(* IEC 61131-3 sources: std_i2980_v2.06_cp053/Source/IMM/ieccontrol/Ejector1, 2 files *)

(* ---- ABMeasure.pu ---- *)
IMPORT_OVER_LISTFILE
 GET_MY_FU_NAME
, KSWO_AddVariable
, WRITE_SVREAL_DIRECT
, FAddToScopeGroup
, KAPPL_LintabData_2P
, KAPPL_MeasureMonitoring
, KSWO_Status
, ABMeasureAI

END_IMPORT

ALGORITHM_BLOCK ABMeasure #DUMMY_EDIT_BLOCK

SYSTEM_VAR
 sv_EjectorLintab : KAPPL_LintabData_2P;
 sv_rEjectorPosition : REAL;
 ai_Position : REAL;
 sv_bTransducerError : BOOL;
 sv_bDeviceReady : BOOL;
 sv_rEjectorVelocity : REAL;
 sv_EjectorMonitorMeas : KAPPL_MeasureMonitoring;
END_VAR

SYSTEM_OBJECT
 TaskAnalog : TASK;
 TaskSlow : TASK;
END_OBJECT

PROCESS_ALGORITHM paInitDebugMeasurement ON TaskSlow AUTOSTART

VAR
 variableName : STRING(255);
 swoState : KSWO_Status;
 b : BOOL;
END_VAR
#BEGIN_EDIT_BLOCK
(**************************************** WARNING ********************************************
 *** The KEBA Kemro K2 System including software is not intended for safety control tasks! ***
 ***                       For further information see Comment tab!                        ***
 *********************************************************************************************)

variableName := CONCAT(GET_MY_FU_NAME(),'.rPosition mm');
swoState := KSWO_AddVariable( Task := TaskAnalog,
                              Name := variableName,
                              Variable := sv_rEjectorPosition);
b := FAddToScopeGroup(Task := TaskAnalog,
                      Name := variableName,
                      GroupId := cScopeGroupEjector);
variableName := CONCAT(GET_MY_FU_NAME(),'.rVelocity mm/s');
swoState := KSWO_AddVariable( Task := TaskAnalog,
                              Name := variableName,
                              Variable := sv_rEjectorVelocity);
b := FAddToScopeGroup(Task := TaskAnalog,
                      Name := variableName,
                      GroupId := cScopeGroupEjector);

STOP_PROCESS_ALGORITHM();

;#END_EDIT_BLOCK END_ALGORITHM

PROCESS_ALGORITHM paMeasure ON TaskAnalog(1000) AUTOSTART

VAR_TEMP
 b : BOOL;
END_VAR

VAR
 abEjectorMeasure : ABMeasureAI;
END_VAR

(* IecGraph-Code *)

(* init step *)
INITIAL_STEP S_Start:
END_STEP

(* steps *)
STEP S_Stop:
AStop (P);
END_STEP

ACTION AStop: #BEGIN_EDIT_BLOCK
STOP_PROCESS_ALGORITHM();

;#END_EDIT_BLOCK END_ACTION (*AStop*)
STEP S_Init:
AInitMeasureBlock (P);
END_STEP

STEP S_Measure:
AMeasure (N);
END_STEP

(* transitions *)
TRANSITION TLinked (* TLinked *) FROM S_Start TO S_Init :=  #BEGIN_EDIT_BLOCK
IS_LINKED(ai_Position)
;#END_EDIT_BLOCK
END_TRANSITION

TRANSITION TNotLinked (* TNotLinked *) FROM S_Start TO S_Stop :=  #BEGIN_EDIT_BLOCK
NOT IS_LINKED(ai_Position)
;#END_EDIT_BLOCK
END_TRANSITION

TRANSITION TStop (* TStop *) FROM S_Stop TO S_Start :=  #BEGIN_EDIT_BLOCK
TRUE
;#END_EDIT_BLOCK
END_TRANSITION

TRANSITION TInitDone (* TInitDone *) FROM S_Init TO S_Measure :=  #BEGIN_EDIT_BLOCK
TRUE
;#END_EDIT_BLOCK
END_TRANSITION

(* end IecGraph-Code *)
(* sfc-code *)

(* stand alone actions *)
ACTION AMeasure: #BEGIN_EDIT_BLOCK
(**************************************** WARNING ********************************************
 *** The KEBA Kemro K2 System including software is not intended for safety control tasks! ***
 ***                       For further information see Comment tab!                        ***
 *********************************************************************************************)

abEjectorMeasure.aRun(bIdle := sv_bDeviceReady);
sv_bTransducerError := abEjectorMeasure.aRun.bSensorError;
b := WRITE_SVREAL_DIRECT(sv_rEjectorPosition, abEjectorMeasure.aRun.rValue);
b := WRITE_SVREAL_DIRECT(sv_rEjectorVelocity, abEjectorMeasure.aRun.rVelocity);

;#END_EDIT_BLOCK END_ACTION (*AMeasure*)
ACTION AInitMeasureBlock: #BEGIN_EDIT_BLOCK
(**************************************** WARNING ********************************************
 *** The KEBA Kemro K2 System including software is not intended for safety control tasks! ***
 ***                       For further information see Comment tab!                        ***
 *********************************************************************************************)

abEjectorMeasure.aInit(sRawValue := 'Ejector1.ai_Position',
                       pLintabPointArray :=  @sv_EjectorLintab.LintabPoints.Point,
                       piUsedLintabPoints := @sv_EjectorLintab.LintabPoints.uNoOfPoints);

abEjectorMeasure.aInitMonitoring(bEnable := sv_EjectorMonitorMeas.EnableMonitoring,
                                 rLowLimit := sv_EjectorMonitorMeas.LowerLimit,
                                 bLimitation := sv_EjectorMonitorMeas.Limitation,
                                 rFailureFactor := sv_EjectorMonitorMeas.FailureFactor);

;#END_EDIT_BLOCK END_ACTION (*AInitMeasureBlock*)
(* end sfc-code *)

END_ALGORITHM

END_ALGORITHM_BLOCK

#END_OF_IEC_PART

@Puma @IecEditor 6 103 @Pou 25
@@@BEG_Comment@@@

@@@END_Comment@@@

@BEG_Contents

@BEG_Func
@RT(17)FuncTreeContainer
4
@Var @RT(14)GET_MY_FU_NAME @RT(0) @T @T @DERIVED 0 @F @RT(22)KEBA_STANDARD_FUNCTION @F
@T
@BEG_Attrib
0 @RT(0) @RT(0)
@END_Attrib
1 1 @F @F @F @F

@Var @RT(16)KSWO_AddVariable @RT(0) @T @T @DERIVED 0 @F @RT(22)KEBA_STANDARD_FUNCTION @F
@T
@BEG_Attrib
0 @RT(0) @RT(0)
@END_Attrib
1 1 @F @F @F @F

@Var @RT(19)WRITE_SVREAL_DIRECT @RT(0) @T @T @DERIVED 0 @F @RT(22)KEBA_STANDARD_FUNCTION @F
@T
@BEG_Attrib
0 @RT(0) @RT(0)
@END_Attrib
1 1 @F @F @F @F

@Var @RT(16)FAddToScopeGroup @RT(0) @T @T @DERIVED 0 @F @RT(8)FUNCTION @F
@T
@BEG_Attrib
0 @RT(0) @RT(0)
@END_Attrib
1 1 @F @F @F @F

@END_Func

@BEG_Const
@RT(18)ConstTreeContainer
0
@END_Const

@BEG_Export

@BEG_Kind
@ALGORITHM_BLOCK @RT(9)ABMeasure @STRUCTURED_TEXT
@RT(0) @RT(0) @RT(0)
@END_Kind

@BEG_Dcl
@RT(16)DclTreeContainer
9
@Var @RT(16)sv_EjectorLintab @RT(0) @T @T @DERIVED 0 @F @RT(19)KAPPL_LintabData_2P @F
@T
@BEG_Attrib
3 @RT(0) @RT(0) @RT(0)
@END_Attrib
1 8 @F @F @F @F

@Var @RT(19)sv_rEjectorPosition @RT(0) @T @F @DT @RT(4)REAL @RT(0) @T @T @BASIC 0 @F
@F @F
@T
@BEG_Attrib
3 @RT(0) @RT(0) @RT(0)
@END_Attrib
1 8 @F @F @F @F

@Var @RT(11)ai_Position @RT(0) @T @F @DT @RT(4)REAL @RT(0) @T @T @BASIC 0 @F
@F @F
@T
@BEG_Attrib
3 @RT(0) @RT(0) @RT(0)
@END_Attrib
1 8 @F @F @F @F

@Var @RT(19)sv_bTransducerError @RT(0) @T @F @DT @RT(4)BOOL @RT(0) @T @T @BASIC 0 @F
@F @F
@T
@BEG_Attrib
3 @RT(0) @RT(0) @RT(0)
@END_Attrib
1 8 @F @F @F @F

@Var @RT(15)sv_bDeviceReady @RT(0) @T @F @DT @RT(4)BOOL @RT(0) @T @T @BASIC 0 @F
@F @F
@T
@BEG_Attrib
3 @RT(0) @RT(0) @RT(0)
@END_Attrib
1 8 @F @F @F @F

@Var @RT(19)sv_rEjectorVelocity @RT(0) @T @F @DT @RT(4)REAL @RT(0) @T @T @BASIC 0 @F
@F @F
@T
@BEG_Attrib
3 @RT(0) @RT(0) @RT(0)
@END_Attrib
1 8 @F @F @F @F

@Var @RT(21)sv_EjectorMonitorMeas @RT(0) @T @T @DERIVED 0 @T @T @DT @RT(23)KAPPL_MeasureMonitoring @RT(0) @T @T @UNKNOWN 0 @F
@F @F
@T
@BEG_Attrib
3 @RT(0) @RT(0) @RT(0)
@END_Attrib
1 8 @F @F @F @F

@Var @RT(10)TaskAnalog @RT(0) @T @F @DT @RT(4)TASK @RT(0) @T @T @BASIC 0 @F
@F @F
@T
@BEG_Attrib
3 @RT(0) @RT(0) @RT(0)
@END_Attrib
1 7 @F @F @F @F

@Var @RT(8)TaskSlow @RT(0) @T @F @DT @RT(4)TASK @RT(0) @T @T @BASIC 0 @F
@F @F
@T
@BEG_Attrib
3 @RT(0) @RT(0) @RT(0)
@END_Attrib
1 7 @F @F @F @F

@END_Dcl

@END_Export

@BEG_Body

2

@BEG_Export

@BEG_Algo
@PROCESS_ALGORITHM @RT(22)paInitDebugMeasurement @STRUCTURED_TEXT
@RT(0) @RT(0) @RT(8)TaskSlow @T @F
@END_Algo

@BEG_Dcl
@RT(16)DclTreeContainer
3
@Var @RT(12)variableName @RT(0) @T @F @DT @RT(11)STRING(255) @RT(0) @T @T @STRING 0 @F @RT(3)255 @F
@F @F
@T
@BEG_Attrib
3 @RT(0) @RT(0) @RT(0)
@END_Attrib
1 0 @F @F @F @F

@Var @RT(8)swoState @RT(0) @T @T @DERIVED 0 @T @T @DT @RT(11)KSWO_Status @RT(0) @T @T @UNKNOWN 0 @F
@F @F
@T
@BEG_Attrib
3 @RT(0) @RT(0) @RT(0)
@END_Attrib
1 0 @F @F @F @F

@Var @RT(1)b @RT(0) @T @F @DT @RT(4)BOOL @RT(0) @T @T @BASIC 0 @F
@F @F
@T
@BEG_Attrib
3 @RT(0) @RT(0) @RT(0)
@END_Attrib
1 0 @F @F @F @F

@END_Dcl

@END_Export

@BEG_Export

@BEG_Algo
@PROCESS_ALGORITHM @RT(9)paMeasure @SEQUENTIAL_FLOW_CHART
@RT(0) @RT(0) @RT(16)TaskAnalog(1000) @T @F
@END_Algo

@BEG_Dcl
@RT(16)DclTreeContainer
2
@Var @RT(16)abEjectorMeasure @RT(0) @T @T @DERIVED 0 @T @T @DT @RT(11)ABMeasureAI @RT(0) @T @T @UNKNOWN 0 @F
@F @F
@T
@BEG_Attrib
3 @RT(0) @RT(0) @RT(0)
@END_Attrib
1 0 @F @F @F @F

@Var @RT(1)b @RT(0) @T @F @DT @RT(4)BOOL @RT(0) @T @T @BASIC 0 @F
@F @F
@T
@BEG_Attrib
3 @RT(0) @RT(0) @RT(0)
@END_Attrib
1 4 @F @F @F @F

@END_Dcl

@END_Export

@BEG_Body
@TL(22)
(**************************************** WARNING ********************************************
 *** The KEBA Kemro K2 System including software is not intended for safety control tasks! ***
 ***                       For further information see Comment tab!                        ***
 *********************************************************************************************)

variableName := CONCAT(GET_MY_FU_NAME(),'.rPosition mm');
swoState := KSWO_AddVariable( Task := TaskAnalog,
                              Name := variableName,
                              Variable := sv_rEjectorPosition);
b := FAddToScopeGroup(Task := TaskAnalog,
                      Name := variableName,
                      GroupId := cScopeGroupEjector);
variableName := CONCAT(GET_MY_FU_NAME(),'.rVelocity mm/s');
swoState := KSWO_AddVariable( Task := TaskAnalog,
                              Name := variableName,
                              Variable := sv_rEjectorVelocity);
b := FAddToScopeGroup(Task := TaskAnalog,
                      Name := variableName,
                      GroupId := cScopeGroupEjector);

STOP_PROCESS_ALGORITHM();

@END_Body

@@@BEG_Comment@@@
@TL(0)

@@@END_Comment@@@

@BEG_SfcBody
4 6 5

@BEG_SfcData 2
@StepSeq @RT(4)sseq @F 5
@Step @RT(7)S_Start @F @T @T @F @RT(0) @F
@AcbCont @RT(7)unnamed @F 0

@AltBranch @RT(3)alt @F 2
@TransSeq @RT(4)tseq @F 1
@Trans @RT(7)TLinked @F @T @F @F @T @T @TL(2)
IS_LINKED(ai_Position)

@RT(7)TLinked @F

@TransSeq @RT(4)tseq @F 4
@Trans @RT(10)TNotLinked @F @T @F @F @T @T @TL(2)
NOT IS_LINKED(ai_Position)

@RT(10)TNotLinked @F
@Step @RT(6)S_Stop @F @F @F @F @RT(0) @F
@AcbCont @RT(7)unnamed @F 1
@Acb @RT(5)AStop @F @T @RT(1)P @RT(0) @F @F @T @TL(2)
STOP_PROCESS_ALGORITHM();

@F

@Trans @RT(5)TStop @F @T @F @F @T @T @TL(2)
TRUE

@RT(5)TStop @F
@Goto @RT(7)S_Start @F @F

@Step @RT(6)S_Init @F @F @F @F @RT(0) @F
@AcbCont @RT(7)unnamed @F 1
@Acb @RT(17)AInitMeasureBlock @F @F @RT(1)P @RT(0) @F @F @F @F

@Trans @RT(9)TInitDone @F @T @F @F @T @T @TL(2)
TRUE

@RT(9)TInitDone @F
@Step @RT(9)S_Measure @F @F @F @F @RT(0) @F
@AcbCont @RT(7)unnamed @F 1
@Acb @RT(8)AMeasure @F @F @RT(1)N @RT(0) @F @F @F @F

@END_SfcData
@SaActions 2
@SaText @RT(8)AMeasure 1 @TL(10)
(**************************************** WARNING ********************************************
 *** The KEBA Kemro K2 System including software is not intended for safety control tasks! ***
 ***                       For further information see Comment tab!                        ***
 *********************************************************************************************)

abEjectorMeasure.aRun(bIdle := sv_bDeviceReady);
sv_bTransducerError := abEjectorMeasure.aRun.bSensorError;
b := WRITE_SVREAL_DIRECT(sv_rEjectorPosition, abEjectorMeasure.aRun.rValue);
b := WRITE_SVREAL_DIRECT(sv_rEjectorVelocity, abEjectorMeasure.aRun.rVelocity);

@SaText @RT(17)AInitMeasureBlock 1 @TL(14)
(**************************************** WARNING ********************************************
 *** The KEBA Kemro K2 System including software is not intended for safety control tasks! ***
 ***                       For further information see Comment tab!                        ***
 *********************************************************************************************)

abEjectorMeasure.aInit(sRawValue := 'Ejector1.ai_Position',
                       pLintabPointArray :=  @sv_EjectorLintab.LintabPoints.Point,
                       piUsedLintabPoints := @sv_EjectorLintab.LintabPoints.uNoOfPoints);

abEjectorMeasure.aInitMonitoring(bEnable := sv_EjectorMonitorMeas.EnableMonitoring,
                                 rLowLimit := sv_EjectorMonitorMeas.LowerLimit,
                                 bLimitation := sv_EjectorMonitorMeas.Limitation,
                                 rFailureFactor := sv_EjectorMonitorMeas.FailureFactor);

@SaTrans 0
@SaExits 0
@END_SfcBody

@@@BEG_Comment@@@
@TL(0)

@@@END_Comment@@@
@END_Body

@END_Contents

(* ---- ABValveControl.pu ---- *)
IMPORT_OVER_LISTFILE
 cMoveBwd
, tsMoveCtrl

END_IMPORT

ALGORITHM_BLOCK ABValveControl #DUMMY_EDIT_BLOCK

SYSTEM_VAR
 do_Forward : BOOL;
 do_Backward : BOOL;
 sv_bFwdActive : BOOL (* Ejector forward is active *);
 sv_bBwdActive : BOOL (* Ejector backward is active *);
 sv_bOutputActive : BOOL (* Output is active *);
 sv_bPreOutputReady : BOOL (* PreOutput is ready *);
END_VAR

SYSTEM_OBJECT
 TaskAnalog : TASK;
END_OBJECT

VAR_EXTERNAL
 g_MoveCtrl : tsMoveCtrl;
END_VAR

PROCESS_ALGORITHM paRun ON TaskAnalog(10001)

VAR
 bFwdStateOld : BOOL;
 bBwdStateOld : BOOL;
END_VAR

(* IecGraph-Code *)

(* init step *)
INITIAL_STEP START:
END_STEP

(* steps *)
STEP Step19:
END_STEP

STEP SET_VALVE_FWD:
ASetFwd (P);
END_STEP

ACTION ASetFwd: #BEGIN_EDIT_BLOCK
do_Forward := TRUE;

;#END_EDIT_BLOCK END_ACTION (*ASetFwd*)
STEP RESET_VALVE_FWD:
AResetFwd (P);
END_STEP

ACTION AResetFwd: #BEGIN_EDIT_BLOCK
do_Forward := FALSE;

;#END_EDIT_BLOCK END_ACTION (*AResetFwd*)
STEP SET_VALVE_BWD:
ASetBwd (P);
END_STEP

ACTION ASetBwd: #BEGIN_EDIT_BLOCK
do_Backward := TRUE;

;#END_EDIT_BLOCK END_ACTION (*ASetBwd*)
STEP RESET_VALVE_BWD:
AResetBwd (P);
END_STEP

ACTION AResetBwd: #BEGIN_EDIT_BLOCK
do_Backward := FALSE;

;#END_EDIT_BLOCK END_ACTION (*AResetBwd*)
STEP SET_VALVE_SHAKE:
ASetShake (P);
END_STEP

ACTION ASetShake: #BEGIN_EDIT_BLOCK
do_Forward := sv_bFwdActive;
do_Backward := sv_bBwdActive;

bFwdStateOld := sv_bFwdActive;
bBwdStateOld := sv_bBwdActive;

;#END_EDIT_BLOCK END_ACTION (*ASetShake*)
STEP Step18:
AResetShake (P);
END_STEP

ACTION AResetShake: #BEGIN_EDIT_BLOCK
do_Forward := FALSE;
do_Backward := FALSE;

;#END_EDIT_BLOCK END_ACTION (*AResetShake*)
STEP END:
Action3 (P);
END_STEP

ACTION Action3: #BEGIN_EDIT_BLOCK
STOP_PROCESS_ALGORITHM();

;#END_EDIT_BLOCK END_ACTION (*Action3*)

(* transitions *)
GO_ON_TRANSITION Trans32 (* Trans32 *) FROM START TO Step19 :=  #BEGIN_EDIT_BLOCK
sv_bPreOutputReady AND
sv_bOutputActive
;#END_EDIT_BLOCK
END_TRANSITION

TRANSITION Trans33 (* Trans33 *) FROM START TO END :=  #BEGIN_EDIT_BLOCK
NOT sv_bOutputActive
;#END_EDIT_BLOCK
END_TRANSITION

GO_ON_TRANSITION Trans1 (* Trans1 *) FROM Step19 TO SET_VALVE_FWD :=  #BEGIN_EDIT_BLOCK
g_MoveCtrl.pData^.MoveId =
cMoveFwd
;#END_EDIT_BLOCK
END_TRANSITION

GO_ON_TRANSITION Trans28 (* Trans28 *) FROM SET_VALVE_FWD TO RESET_VALVE_FWD :=  #BEGIN_EDIT_BLOCK
NOT sv_bOutputActive
;#END_EDIT_BLOCK
END_TRANSITION

GO_ON_TRANSITION Trans17 (* Trans17 *) FROM RESET_VALVE_FWD TO END :=  #BEGIN_EDIT_BLOCK
TRUE
;#END_EDIT_BLOCK
END_TRANSITION

GO_ON_TRANSITION Trans3 (* Trans3 *) FROM Step19 TO SET_VALVE_BWD :=  #BEGIN_EDIT_BLOCK
g_MoveCtrl.pData^.MoveId =
cMoveBwd
;#END_EDIT_BLOCK
END_TRANSITION

GO_ON_TRANSITION Trans6 (* Trans6 *) FROM SET_VALVE_BWD TO RESET_VALVE_BWD :=  #BEGIN_EDIT_BLOCK
NOT sv_bOutputActive
;#END_EDIT_BLOCK
END_TRANSITION

GO_ON_TRANSITION Trans18 (* Trans18 *) FROM RESET_VALVE_BWD TO END :=  #BEGIN_EDIT_BLOCK
TRUE
;#END_EDIT_BLOCK
END_TRANSITION

GO_ON_TRANSITION Trans31 (* Trans31 *) FROM Step19 TO SET_VALVE_SHAKE :=  #BEGIN_EDIT_BLOCK
g_MoveCtrl.pData^.MoveId =
cMoveShake
;#END_EDIT_BLOCK
END_TRANSITION

TRANSITION Trans34 (* Trans34 *) FROM SET_VALVE_SHAKE TO SET_VALVE_SHAKE :=  #BEGIN_EDIT_BLOCK
bFwdStateOld <> sv_bFwdActive OR
bBwdStateOld <> sv_bBwdActive

;#END_EDIT_BLOCK
END_TRANSITION

GO_ON_TRANSITION Trans39 (* Trans33 *) FROM SET_VALVE_SHAKE TO Step18 :=  #BEGIN_EDIT_BLOCK
NOT sv_bOutputActive
;#END_EDIT_BLOCK
END_TRANSITION

GO_ON_TRANSITION Trans54 (* Trans32 *) FROM Step18 TO END :=  #BEGIN_EDIT_BLOCK
TRUE
;#END_EDIT_BLOCK
END_TRANSITION

TRANSITION Trans30 (* Trans30 *) FROM Step19 TO END :=  #BEGIN_EDIT_BLOCK
NOT sv_bOutputActive
;#END_EDIT_BLOCK
END_TRANSITION

TRANSITION Trans16 (* Trans16 *) FROM END TO START :=  #BEGIN_EDIT_BLOCK
TRUE
;#END_EDIT_BLOCK
END_TRANSITION

(* end IecGraph-Code *)
(* sfc-code *)
(* end sfc-code *)

END_ALGORITHM

POSTUPDATE_ALGORITHM pOutputActive ON TaskAnalog(10000) WITH sv_bOutputActive

#BEGIN_EDIT_BLOCK
IF sv_bOutputActive THEN

    START_PROCESS_ALGORITHM(paRun);
END_IF;

;#END_EDIT_BLOCK END_ALGORITHM

END_ALGORITHM_BLOCK

#END_OF_IEC_PART

@Puma @IecEditor 6 97 @Pou 25
@@@BEG_Comment@@@

@@@END_Comment@@@

@BEG_Contents

@BEG_Func
@RT(17)FuncTreeContainer
0
@END_Func

@BEG_Const
@RT(18)ConstTreeContainer
1
@Var @RT(8)cMoveBwd @RT(0) @T @F @DT @RT(4)DINT @RT(0) @T @T @BASIC 0 @F
@F @F
@T
@BEG_Attrib
0 @RT(2)11 @RT(17)movement backward
@END_Attrib
1 1 @F @F @F @F

@END_Const

@BEG_Export

@BEG_Kind
@ALGORITHM_BLOCK @RT(14)ABValveControl @STRUCTURED_TEXT
@RT(0) @RT(0) @RT(0)
@END_Kind

@BEG_Dcl
@RT(16)DclTreeContainer
8
@Var @RT(10)g_MoveCtrl @RT(0) @T @T @DERIVED 0 @T @T @DT @RT(10)tsMoveCtrl @RT(0) @T @T @UNKNOWN 0 @F
@F @F
@T
@BEG_Attrib
3 @RT(0) @RT(0) @RT(0)
@END_Attrib
1 6 @F @F @F @F

@Var @RT(10)do_Forward @RT(0) @T @F @DT @RT(4)BOOL @RT(0) @T @T @BASIC 0 @F
@F @F
@T
@BEG_Attrib
3 @RT(0) @RT(0) @RT(0)
@END_Attrib
1 8 @F @F @F @F

@Var @RT(11)do_Backward @RT(0) @T @F @DT @RT(4)BOOL @RT(0) @T @T @BASIC 0 @F
@F @F
@T
@BEG_Attrib
3 @RT(0) @RT(0) @RT(0)
@END_Attrib
1 8 @F @F @F @F

@Var @RT(13)sv_bFwdActive @RT(0) @T @F @DT @RT(4)BOOL @RT(0) @T @T @BASIC 0 @F
@F @F
@T
@BEG_Attrib
3 @RT(0) @RT(25)Ejector forward is active @RT(0)
@END_Attrib
1 8 @F @F @F @F

@Var @RT(13)sv_bBwdActive @RT(0) @T @F @DT @RT(4)BOOL @RT(0) @T @T @BASIC 0 @F
@F @F
@T
@BEG_Attrib
3 @RT(0) @RT(26)Ejector backward is active @RT(0)
@END_Attrib
1 8 @F @F @F @F

@Var @RT(16)sv_bOutputActive @RT(0) @T @F @DT @RT(4)BOOL @RT(0) @T @T @BASIC 0 @F
@F @F
@T
@BEG_Attrib
3 @RT(0) @RT(16)Output is active @RT(0)
@END_Attrib
1 8 @F @F @F @F

@Var @RT(18)sv_bPreOutputReady @RT(0) @T @F @DT @RT(4)BOOL @RT(0) @T @T @BASIC 0 @F
@F @F
@T
@BEG_Attrib
3 @RT(0) @RT(18)PreOutput is ready @RT(0)
@END_Attrib
1 8 @F @F @F @F

@Var @RT(10)TaskAnalog @RT(0) @T @T @RENAMED 0 @T @T @DT @RT(4)TASK @RT(0) @T @T @BASIC 0 @F
@F @F
@T
@BEG_Attrib
3 @RT(0) @RT(0) @RT(0)
@END_Attrib
1 7 @F @F @F @F

@END_Dcl

@END_Export

@BEG_Body

2

@BEG_Export

@BEG_Algo
@PROCESS_ALGORITHM @RT(5)paRun @SEQUENTIAL_FLOW_CHART
@RT(0) @RT(0) @RT(17)TaskAnalog(10001) @F @F
@END_Algo

@BEG_Dcl
@RT(16)DclTreeContainer
2
@Var @RT(12)bFwdStateOld @RT(0) @T @F @DT @RT(4)BOOL @RT(0) @T @T @BASIC 0 @F
@F @F
@T
@BEG_Attrib
3 @RT(0) @RT(0) @RT(0)
@END_Attrib
1 0 @F @F @F @F

@Var @RT(12)bBwdStateOld @RT(0) @T @F @DT @RT(4)BOOL @RT(0) @T @T @BASIC 0 @F
@F @F
@T
@BEG_Attrib
3 @RT(0) @RT(0) @RT(0)
@END_Attrib
1 0 @F @F @F @F

@END_Dcl

@END_Export

@BEG_Export

@BEG_Algo
@POSTUPDATE_ALGORITHM @RT(13)pOutputActive @STRUCTURED_TEXT
@RT(0) @RT(16)sv_bOutputActive @RT(17)TaskAnalog(10000) @F @F
@END_Algo

@BEG_Dcl
@RT(16)DclTreeContainer
0
@END_Dcl

@END_Export

@BEG_SfcBody
21 20 35

@BEG_SfcData 2
@StepSeq @RT(4)sseq @F 1
@Loop @RT(4)loop @F 2
@StepSeq @RT(3)seq @F 5
@Step @RT(5)START @F @T @F @F @RT(0) @F
@AcbCont @RT(7)unnamed @F 0

@AltBranch @RT(3)alt @F 2
@TransSeq @RT(4)tseq @F 1
@Trans @RT(7)Trans32 @F @T @F @F @T @F @TL(3)
sv_bPreOutputReady AND
sv_bOutputActive

@RT(7)Trans32 @F

@TransSeq @RT(4)tseq @F 2
@Trans @RT(7)Trans33 @F @T @F @F @T @T @TL(2)
NOT sv_bOutputActive

@RT(7)Trans33 @F
@Goto @RT(3)END @F @F

@Step @RT(6)Step19 @F @F @F @F @RT(0) @F
@AcbCont @RT(7)unnamed @F 0

@AltBranch @RT(3)alt @F 4
@TransSeq @RT(4)tseq @F 5
@Trans @RT(6)Trans1 @F @T @F @F @T @F @TL(3)
g_MoveCtrl.pData^.MoveId =
cMoveFwd

@RT(6)Trans1 @F
@Step @RT(13)SET_VALVE_FWD @F @F @F @F @RT(0) @F
@AcbCont @RT(7)unnamed @F 1
@Acb @RT(7)ASetFwd @F @T @RT(1)P @RT(0) @F @F @T @TL(2)
do_Forward := TRUE;

@F

@Trans @RT(7)Trans28 @F @T @F @F @T @F @TL(2)
NOT sv_bOutputActive

@RT(7)Trans28 @F
@Step @RT(15)RESET_VALVE_FWD @F @F @F @F @RT(0) @F
@AcbCont @RT(7)unnamed @F 1
@Acb @RT(9)AResetFwd @F @T @RT(1)P @RT(0) @F @F @T @TL(2)
do_Forward := FALSE;

@F

@Trans @RT(7)Trans17 @F @T @F @F @T @F @TL(2)
TRUE

@RT(7)Trans17 @F

@TransSeq @RT(4)tseq @F 5
@Trans @RT(6)Trans3 @F @T @F @F @T @F @TL(3)
g_MoveCtrl.pData^.MoveId =
cMoveBwd

@RT(6)Trans3 @F
@Step @RT(13)SET_VALVE_BWD @F @F @F @F @RT(0) @F
@AcbCont @RT(7)unnamed @F 1
@Acb @RT(7)ASetBwd @F @T @RT(1)P @RT(0) @F @F @T @TL(2)
do_Backward := TRUE;

@F

@Trans @RT(6)Trans6 @F @T @F @F @T @F @TL(2)
NOT sv_bOutputActive

@RT(6)Trans6 @F
@Step @RT(15)RESET_VALVE_BWD @F @F @F @F @RT(0) @F
@AcbCont @RT(7)unnamed @F 1
@Acb @RT(9)AResetBwd @F @T @RT(1)P @RT(0) @F @F @T @TL(2)
do_Backward := FALSE;

@F

@Trans @RT(7)Trans18 @F @T @F @F @T @F @TL(2)
TRUE

@RT(7)Trans18 @F

@TransSeq @RT(4)tseq @F 5
@Trans @RT(7)Trans31 @F @T @F @F @T @F @TL(3)
g_MoveCtrl.pData^.MoveId =
cMoveShake

@RT(7)Trans31 @F
@Loop @RT(4)loop @F 2
@StepSeq @RT(3)seq @F 1
@Step @RT(15)SET_VALVE_SHAKE @F @F @F @F @RT(0) @F
@AcbCont @RT(7)unnamed @F 1
@Acb @RT(9)ASetShake @F @T @RT(1)P @RT(0) @F @F @T @TL(6)
do_Forward := sv_bFwdActive;
do_Backward := sv_bBwdActive;

bFwdStateOld := sv_bFwdActive;
bBwdStateOld := sv_bBwdActive;

@F

@Trans @RT(7)Trans34 @F @T @T @T @T @T @TL(4)
bFwdStateOld <> sv_bFwdActive OR
bBwdStateOld <> sv_bBwdActive

@RT(7)Trans34 @F

@Trans @RT(7)Trans39 @F @T @F @F @T @F @TL(2)
NOT sv_bOutputActive

@RT(7)Trans33 @F
@Step @RT(6)Step18 @F @F @F @F @RT(0) @F
@AcbCont @RT(7)unnamed @F 1
@Acb @RT(11)AResetShake @F @T @RT(1)P @RT(0) @F @F @T @TL(3)
do_Forward := FALSE;
do_Backward := FALSE;

@F

@Trans @RT(7)Trans54 @F @T @F @F @T @F @TL(2)
TRUE

@RT(7)Trans32 @F

@TransSeq @RT(4)tseq @F 2
@Trans @RT(7)Trans30 @F @T @F @F @T @T @TL(2)
NOT sv_bOutputActive

@RT(7)Trans30 @F
@Goto @RT(3)END @F @F

@Step @RT(3)END @F @F @T @F @RT(0) @F
@AcbCont @RT(7)unnamed @F 1
@Acb @RT(7)Action3 @F @T @RT(1)P @RT(0) @F @F @T @TL(2)
STOP_PROCESS_ALGORITHM();

@F

@Trans @RT(7)Trans16 @F @T @T @T @T @T @TL(2)
TRUE

@RT(7)Trans16 @F

@END_SfcData
@SaActions 0
@SaTrans 0
@SaExits 0
@END_SfcBody

@@@BEG_Comment@@@
@TL(0)

@@@END_Comment@@@

@BEG_Body
@TL(5)
IF sv_bOutputActive THEN

    START_PROCESS_ALGORITHM(paRun);
END_IF;

@END_Body

@@@BEG_Comment@@@
@TL(0)

@@@END_Comment@@@
@END_Body

@END_Contents
